FUNCTION_BLOCK F_RIGHT (* rightmost L characters of IN *)
  (* Standard: 61131-3; Classification: standard character and string function; Description: Copyright (c) 2013 TU Wien ACIN This program and the accompanying materials are made available under the terms of the Eclipse Public License 2.0 which is available at https://www.eclipse.org/legal/epl-2.0/ SPDX-License-Identifier: EPL-2.0 *)
  (* Version 1.0, 2013-08-27, Monika Wenger, TU Wien ACIN *)
  (* Version 3.0, 2025-04-14, Patrick Aigner, changed package *)
  PACKAGE iec61131::charString;
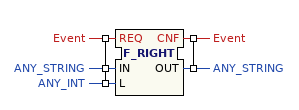
  EVENT_INPUT
    REQ WITH IN, L; (* Service Request *)
  END_EVENT
  EVENT_OUTPUT
    CNF WITH OUT; (* Confirmation of Requested Service *)
  END_EVENT
  VAR_INPUT
    IN : ANY_STRING; (* input string *)
    L : ANY_INT; (* sub-string start position *)
  END_VAR
  VAR_OUTPUT
    OUT : ANY_STRING; (* sub-string from L to string length *)
  END_VAR
END_FUNCTION_BLOCK
